FUNCTION_BLOCK AX_TOF (* standard timer function block (off-delay timing) *)
  (* Standard: 61499-2; Classification: standard timer function block; Description: Copyright (c) 2024 HR Agrartechnik GmbH This program and the accompanying materials are made available under the terms of the Eclipse Public License 2.0 which is available at https://www.eclipse.org/legal/epl-2.0/ SPDX-License-Identifier: EPL-2.0 *)
  (* Version 3.0, 2025-04-14, Patrick Aigner, changed package *)
  (* Version 1.1, 2024-04-23, Franz Höpfinger, HR Agrartechnik GmbH, Add a Reset to Timer FBs *)
  (* Version 1.0, 2024-03-04, Franz Höpfinger, HR Agrartechnik GmbH *)
  PACKAGE adapter::events::unidirectional::timers;
  IMPORT eclipse4diac::core::TypeHash;
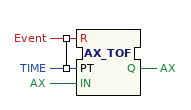
  EVENT_INPUT
    R WITH PT; (* Reset *)
  END_EVENT
  VAR_INPUT
    PT : TIME; (* Process time *)
  END_VAR
  SOCKETS
    IN : adapter::types::unidirectional::AX; (* Input *)
  END_SOCKETS
  PLUGS
    Q : adapter::types::unidirectional::AX; (* Output *)
  END_PLUGS
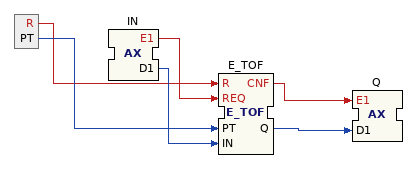
  FBS
    E_TOF : iec61499::events::timers::E_TOF;
  END_FBS
  EVENT_CONNECTIONS
    R TO E_TOF.R;
    E_TOF.CNF TO Q.E1;
    IN.E1 TO E_TOF.REQ;
  END_CONNECTIONS
  DATA_CONNECTIONS
    PT TO E_TOF.PT;
    E_TOF.Q TO Q.D1;
    IN.D1 TO E_TOF.IN;
  END_CONNECTIONS
END_FUNCTION_BLOCK
